(* IEC 61131-3 sources: AXOpen/src/templates.simple/app/src/templates/unit, 4 files *)

(* ---- AutomatSequence.st ---- *)
NAMESPACE axosimple.UnitTemplate
    USING axosimple;
    USING AXOpen.Data;
    USING AXOpen.Core;
    USING System.Strings;

    ///<summary>
    /// Provides automatic mode sequence.
    ///</summary>
    {#ix-set:AttributeName = "<#AUTOMAT#>"}
    CLASS PUBLIC AutomatSequence
        EXTENDS AXOpen.Core.AxoSequencerContainer
        VAR PUBLIC
            Steps : ARRAY[0..150] OF AxoStep;
        END_VAR
        VAR PRIVATE
            Components : REF_TO Components;
            ProcessData : REF_TO ProcessDataManger;
            _currentId : STRING;
        END_VAR

        METHOD INTERNAL Run
            VAR_INPUT
                _components : REF_TO Components;
                _processData : REF_TO ProcessDataManger;
                _parent : IAxoObject;
            END_VAR
            Components := _components;
            ProcessData := _processData;
            SUPER.Run(_parent);
        END_METHOD
        ///<summary>
        /// Contains logic of the steps of this sequence
        ///</summary>

        METHOD OVERRIDE Main
            IF (Components = NULL OR ProcessData = NULL) THEN
                RETURN;
            END_IF;

            // This sequecner executes the steps in cycles from top to bottom
            // in the same order they are written in the program
            // Each step in the sequence must can be used only once.
            // This sets the sequence to run in cycles (top-botton-top and again).
            THIS.SequenceMode := eAxoSequenceMode#Cyclic;

            IF (Steps[0].Execute(THIS, TRUE, '<#GET ID#>')) THEN
                //-------------------------------------------------------
                _currentId := '1';
                //-------------------------------------------------------
            END_IF;

            IF (Steps[1].Execute(THIS, TRUE, '<#GET DATA#>')) THEN
                //-------------------------------------------------------
                IF (ProcessData^.Read(_currentId).IsDone()) THEN
                    THIS.MoveNext();
                END_IF;
                //-------------------------------------------------------
            END_IF;

            IF (Steps[2].Execute(THIS, TRUE, '<#DO SOMETHING#>')) THEN
                //-------------------------------------------------------
                    THIS.MoveNext();
                //-------------------------------------------------------
            END_IF;

            IF (Steps[149].Execute(THIS, TRUE, '<#UPDATE DATA#>')) THEN
                //-------------------------------------------------------
                IF (ProcessData^.Update(_currentId).IsDone()) THEN
                    THIS.MoveNext();
                END_IF;
                //-------------------------------------------------------
            END_IF;

            // This will close the sequence and will return to the first step.
            THIS.Close(Steps[150]);
        END_METHOD
    END_CLASS
END_NAMESPACE

(* ---- Comonents.st ---- *)
NAMESPACE axosimple.UnitTemplate
    USING axosimple;
    USING AXOpen.Data;
    USING AXOpen.Core;
    USING System.Strings;

    ///<summary>
    /// Groups components of this controller unit.
    ///</summary>
    CLASS Components
        EXTENDS AXOpen.Core.AxoObject
        VAR PUBLIC
            // HERE DECLARE COMPONENTS USED BY THIS CONTROLLED UNIT
            // HorizontalCylinder : AXOpen.Components.Pneumatics.AxoCylinder;
            // VerticalCylinder : AXOpen.Components.Pneumatics.AxoCylinder;
            // GripperCylinder : AXOpen.Components.Pneumatics.AxoCylinder;
            // DMCReader : AXOpen.Components.Cognex.Vision.v_6_0_0_0.AxoDataman;
            // PartPresenceSensor : AXOpen.Elements.AxoDi;
        END_VAR

        METHOD PUBLIC Update
            VAR_INPUT
                parent : IAxoObject;
            END_VAR
            VAR_IN_OUT
                Inputs : axosimple.Inputs;
                Outputs : axosimple.Outputs;
            END_VAR
            THIS.Initialize(parent);
            // HERE INITIALIZE YOUR COMPONENTS
            // HorizontalCylinder.Run(THIS, Inputs.B0[0], Inputs.B0[1], Outputs.B0[0], Outputs.B0[1]);
            // VerticalCylinder.Run(THIS, Inputs.B0[2], Inputs.B0[3], Outputs.B0[2], Outputs.B0[3]);
            // GripperCylinder.Run(THIS, Inputs.B0[4], Inputs.B0[5], Outputs.B0[4], Outputs.B0[5]);

        END_METHOD
    END_CLASS
END_NAMESPACE

(* ---- GroundSequence.st ---- *)
NAMESPACE axosimple.UnitTemplate
    USING axosimple;
    USING AXOpen.Data;
    USING AXOpen.Core;
    USING System.Strings;

    ///<summary>
    /// Provides ground mode sequence.
    ///</summary>
    {#ix-set:AttributeName = "<#GROUND#>"}
    CLASS PUBLIC GroundSequence
        EXTENDS AXOpen.Core.AxoSequencerContainer
        VAR PUBLIC
            Steps : ARRAY[0..20] OF AxoStep;
            MoveToWork : AxoTask;
        END_VAR
        VAR PRIVATE
            Components : REF_TO Components;
            ProcessData : REF_TO ProcessDataManger;
            _currentId : STRING;
        END_VAR

        METHOD INTERNAL Run
            VAR_INPUT
                _components : REF_TO Components;
                _processData : REF_TO ProcessDataManger;
                _parent : IAxoObject;
            END_VAR
            Components := _components;
            ProcessData := _processData;
            SUPER.Run(_parent);

            // MoveToWork.Initialize(THIS);

        END_METHOD
        ///<summary>
        /// Contains logic of the steps of this sequence
        ///</summary>

        METHOD PROTECTED OVERRIDE Main
            // IF (Components = NULL OR ProcessData = NULL) THEN
            //     RETURN;
            // END_IF;
            // This sequecner executes the steps in cycles from top to bottom
            // in the same order they are written in the program
            // Each step in the sequence must can be used only once.
            // This sets the sequence to run once (top-botton) and stops with done after closing.
            THIS.SequenceMode := eAxoSequenceMode#RunOnce;
            // This is more verbose but also more versatile way of executing step logic.
            IF (Steps[0].Execute(THIS, TRUE, '<#GET ID#>')) THEN
                //-------------------------------------------------------
                        _currentId := '1';
                        THIS.MoveNext();
                //-------------------------------------------------------
                END_IF;

                IF (Steps[1].Execute(THIS, TRUE, '<#GET DATA#>')) THEN
                //-------------------------------------------------------
                    IF(ProcessData^.Read(_currentId).IsDone()) THEN
                        THIS.MoveNext();
                    END_IF;
                //-------------------------------------------------------
                END_IF;

                IF (Steps[2].Execute(THIS, TRUE, '<#DO SOMETHING#>')) THEN
                    //-------------------------------------------------------
                        THIS.MoveNext();
                    //-------------------------------------------------------
                END_IF;

                IF (Steps[19].Execute(THIS, TRUE, '<#SAVE DATA#>')) THEN
                    //-------------------------------------------------------

                        IF(ProcessData^.Update(_currentId).IsDone()) THEN
                            THIS.MoveNext();
                        END_IF;
                    //-------------------------------------------------------
                END_IF;

            // This will close the sequence and will return to the first step.
            THIS.Close(Steps[20]);
        END_METHOD
    END_CLASS
END_NAMESPACE

(* ---- ServiceMode.st ---- *)
NAMESPACE axosimple.UnitTemplate
    USING axosimple;
    USING AXOpen.Data;
    USING AXOpen.Core;
    USING System.Strings;

    ///<summary>
    /// Provides logic for service/manual/maintenance mode.
    ///</summary>
    {#ix-set:AttributeName = "<#SERVICE#>"}
    CLASS PUBLIC ServiceMode
        EXTENDS AXOpen.Core.AxoTask
        ///<summary>
        /// Runs service mode logic. This method must be called cyclically.
        ///</summary>

        METHOD PUBLIC Run
            VAR_INPUT
                parent : IAxoObject;
            END_VAR
            VAR_IN_OUT
                components : Components;
            END_VAR
            THIS.Initialize(parent);
            IF THIS.Execute() THEN
                THIS.Handle(components);
            END_IF;
        END_METHOD

        METHOD PRIVATE Handle
            VAR_IN_OUT
                components : Components;
            END_VAR
            ;
            // HERE CALL LOGIC FOR MANUAL/SERICE OPERATIONS
            // components.HorizontalCylinder.ActivateManualControl();
            // components.VerticalCylinder.ActivateManualControl();
            // components.GripperCylinder.ActivateManualControl();
        END_METHOD
    END_CLASS
END_NAMESPACE
